TYPE UDT_FaultLogItem :
STRUCT
	stFault 	: UDT_Fault;
	Id			: STRING; // Fault ID used for reporting and checking duplicates (not an unique value unless description matches as well)
	StartTime	: DATE_AND_TIME; // Time the fault became active
	EndTime		: DATE_AND_TIME; // Time the fault stopped being active
END_STRUCT
END_TYPE

(* stored: Version 1.1.0.1, ProductVersion 3.1.4024.11
   DUT UDT_FaultLogItem: Id {10af48dd-fc8f-013a-0221-b64173b2a737} *)
